FUNCTION_BLOCK FB_SK_StateManager

VAR
	bStartUpDone		: BOOL;	
	bFirstAbortDone		: BOOL;
	
	eCommand			: E_XMotion_Command;	
	eCommandOld			: E_XMotion_Command;
	eStatus				: E_XMotion_Status;	
	nCommandCounter		: UDINT;

END_VAR

METHOD PUBLIC Cycle
VAR_INPUT
END_VAR


	IF NOT bStartUpDone THEN					
		eStatus := E_XMotion_Status.StartUp;
	ELSIF NOT bFirstAbortDone THEN
		eStatus := E_XMotion_Status.Aborting;
	ELSE

		IF eCommand <> eCommandOld THEN
			eCommandOld := eCommand;
	
			nCommandCounter := nCommandCounter +1;
			
			
			CASE eCommand OF
				
			
			E_XMotion_Command.Abort:	
						eStatus := E_XMotion_Status.Aborting;	
			
			E_XMotion_Command.Reset:
						IF eStatus = E_XMotion_Status.Aborted THEN
							eStatus := E_XMotion_Status.Resetting;	
						END_IF
				
			E_XMotion_Command.Prepare:
						IF eStatus = E_XMotion_Status.Stopped THEN
							eStatus := E_XMotion_Status.Preparing;	
						END_IF	
			
			E_XMotion_Command.Start:
						IF eStatus = E_XMotion_Status.Prepared THEN
							eStatus := E_XMotion_Status.Execute;	
						END_IF	

			E_XMotion_Command.HoldOnError:
						eStatus := E_XMotion_Status.HoldOnError;

					
			END_CASE
		END_IF
		
	END_IF
END_METHOD

METHOD PUBLIC StateComplete : BOOL
VAR_INPUT
END_VAR




	CASE eStatus OF
		
	E_XMotion_Status.StartUp:
				bStartUpDone := TRUE;
				
	E_XMotion_Status.Aborting:
				bFirstAbortDone := TRUE;	
				eStatus := E_XMotion_Status.Aborted;	
	
	E_XMotion_Status.Resetting:
				eStatus := E_XMotion_Status.Stopped;
		
	E_XMotion_Status.Preparing:
				eStatus := E_XMotion_Status.Prepared;
	
				
	END_CASE
END_METHOD

PROPERTY Status : E_XMotion_Status
GET
Status := eStatus;
END_GET
END_PROPERTY

PROPERTY XMotionCommand : E_XMotion_Command
SET
eCommand := XMotionCommand;
END_SET
END_PROPERTY

END_FUNCTION_BLOCK

(* stored: Version 1.1.0.1, ProductVersion 3.1.4024.9
   POU FB_SK_StateManager: Id {b50383f9-c421-4744-8028-ae8d88a68bff}, SpecialFunc None
   Method Cycle: Id {b55ec817-8381-4105-8024-e51681504619}
   Method StateComplete: Id {4028cc9d-cb45-4cdb-adc3-6e745daebc8d}
   Property Status: Id {08773a9d-3e92-4f76-822b-ff8c7dd0cab9}
   Get Get: Id {b7aa7ae1-1139-4f97-9264-193f48a2ef87}
   Property XMotionCommand: Id {8b04df2b-3437-44f8-b280-10920a7d4b1a}
   Set Set: Id {a90f7e29-ae12-4fd1-a0ae-d9a73140d215} *)
